// TIA Portal V15 export
// export: Created 2018-05-31T14:49:00.3360138Z, ExportSetting WithDefaults, WithReadOnly, DisplayName Totally Integrated Automation Portal, DisplayVersion V15, DisplayName STEP 7 Professional, DisplayVersion V15, DisplayName WinCC Professional, DisplayVersion V15, DisplayName TIA Portal Openness, DisplayVersion V15
DATA_BLOCK "T105"   // DB9
{ S7_Optimized_Access := 'FALSE' }
VERSION : 0.1
// stored: AutoNumber true, CodeModifiedDate 2018-05-31T14:48:47.2782669Z, CompileDate 2018-05-31T14:48:47.7282927Z, CreationDate 2018-05-31T14:47:07.2805474Z, InstanceOfType FB, InterfaceModifiedDate 2018-05-31T08:09:02.725429Z, IsConsistent true, IsKnowHowProtected false, ModifiedDate 2018-05-31T14:48:47.2782669Z, ParameterModified 2018-05-31T08:09:02.725429Z, StructureModified 2018-05-31T08:09:02.725429Z, UDAEnableTagReadback false
BEGIN
END_DATA_BLOCK
